///EL1819 | HD EtherCAT Terminals, 16-channel digital input 24 V DC, 10 µs
FUNCTION_BLOCK EL1819

VAR_INPUT
    En              : BOOL;
    iTerminal_ID    : INT;
    ErrorSystem     : POINTER TO ST_ErrorSystem;
END_VAR

VAR_OUTPUT
    EnO         : BOOL;
    bError      : BOOL;
END_VAR

VAR
    WcState_WcState     AT %I*  : BOOL;
    InfoData_State      AT %I*  : UINT;

    //FB-s
    EL1819_Error    : FB_TerminalError;
END_VAR

(*
* TODO: DONE!
*)
EnO:=En;

//Error FB instance
EL1819_Error(
    En                  := TRUE,
    iTerminal_ID        := iTerminal_ID,
    bWcState            := WcState_WcState,
    uiInfoData_State    := InfoData_State,
    pErrorSystem        := ErrorSystem,
    bError              => bError,
);

END_FUNCTION_BLOCK

(* stored: Version 1.1.0.1, ProductVersion 3.1.4024.0
   POU EL1819: Id {00fa0d24-98b5-49bc-bf41-0a4a34b46bc9}, SpecialFunc None *)
